SUBAPPLICATION Uebung_217b_AX (* Standard IEC 61131-3 ALI_FB_CTD (Adapter Version, LINT) mit Terminal-Ausgabe (PHYS) *)
  (* Standard: 61131-3; Description: Copyright (c) 2026 Meisterschulen am Ostbahnhof This program and the accompanying materials are made available under the terms of the Eclipse Public License 2.0 which is available at https://www.eclipse.org/legal/epl-2.0/ SPDX-License-Identifier: EPL-2.0 *)
  (* Version 1.1, 2026-04-21, Franz Höpfinger, Meisterschulen am Ostbahnhof, Added terminal output for counter value (PHYS) *)
  (* Version 1.0, 2026-04-21, Franz Höpfinger, Meisterschulen am Ostbahnhof, initial API and implementation (Adapter version) *)
  PACKAGE Uebungen;
  IMPORT Uebungen::const::UT::DefaultPool_Numeric::OutputNumber_N3;
  IMPORT logiBUS::io::DI::logiBUS_DI::Input_I1;
  IMPORT logiBUS::io::DI::logiBUS_DI::Input_I2;
  IMPORT logiBUS::io::DQ::logiBUS_DO::Output_Q1;
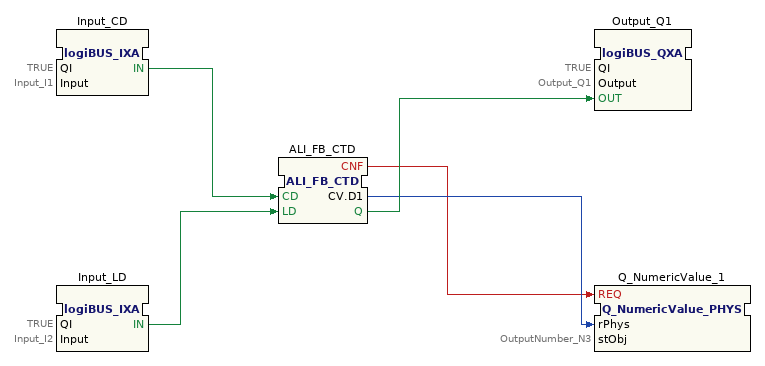
  FBS
    ALI_FB_CTD : adapter::iec61131_3::counters::ALI_FB_CTD;
    Input_CD : logiBUS::io::DI::logiBUS_IXA(QI := TRUE, Input := Input_I1);
    Input_LD : logiBUS::io::DI::logiBUS_IXA(QI := TRUE, Input := Input_I2);
    Output_Q1 : logiBUS::io::DQ::logiBUS_QXA(QI := TRUE, Output := Output_Q1);
    Q_NumericValue_1 : isobus::UT::Q::Q_NumericValue_PHYS(stObj := OutputNumber_N3);
  END_FBS
  EVENT_CONNECTIONS
    ALI_FB_CTD.CNF TO Q_NumericValue_1.REQ;
  END_CONNECTIONS
  DATA_CONNECTIONS
    ALI_FB_CTD.CV.D1 TO Q_NumericValue_1.rPhys;
  END_CONNECTIONS
  ADAPTER_CONNECTIONS
    Input_CD.IN TO ALI_FB_CTD.CD;
    Input_LD.IN TO ALI_FB_CTD.LD;
    ALI_FB_CTD.Q TO Output_Q1.OUT;
  END_CONNECTIONS
END_SUBAPPLICATION
